INTERFACE ITF_SaMController EXTENDS ITF_BaseControlElement, ITF_SaMControllerConfigure, ITF_SaMControllerCommandChange, ITF_BaseSaM

METHOD Execute : BOOL
VAR_INPUT
	iNumberOfCommand		: INT;
	eChangeCategory			: E_SaMChangeCategory;
END_VAR
END_METHOD

METHOD ExecuteTopElementOperationsForCurrentState : BOOL
VAR_INPUT
	itfTopElement				: ITF_BaseSaMStateMethod;
END_VAR
END_METHOD

METHOD PUBLIC ExitActivState
VAR_INPUT
END_VAR
END_METHOD

METHOD PUBLIC GetActiveModeName : ST_BaseLabel
VAR_INPUT
END_VAR
END_METHOD

METHOD PUBLIC GetActiveStateName : ST_BaseLabel
VAR_INPUT
END_VAR
END_METHOD

METHOD PUBLIC GetMode : E_BaseMachineMode
VAR_INPUT
END_VAR
END_METHOD

METHOD PUBLIC GetModeName : ST_BaseLabel
VAR_INPUT
	iNumber			: INT;
END_VAR
END_METHOD

METHOD PUBLIC GetState : E_BaseMachineState
VAR_INPUT
END_VAR
END_METHOD

METHOD GetStateName : ST_BaseLabel
VAR_INPUT
	iNumber			: INT;
END_VAR
END_METHOD

METHOD PUBLIC GetTimeStateForCurrentMode : LTIME
VAR_INPUT
	iNumber		: INT;
END_VAR
END_METHOD

METHOD PUBLIC GetTimeStateForMode : LTIME
VAR_INPUT
	iMode		: int;
	iState		: INT;
END_VAR
END_METHOD

METHOD PUBLIC GetTimeWorkForMode : LTIME
VAR_INPUT
	iMode	: INT;
END_VAR
END_METHOD

METHOD PUBLIC IncrementTimeStateAndMode
VAR_INPUT
	tInterval				: TIME := T#100MS;
END_VAR
END_METHOD

METHOD PUBLIC IsChangeModeBusy : BOOL
VAR_INPUT
END_VAR
END_METHOD

METHOD PUBLIC IsChangeModeDone : BOOL
VAR_INPUT
END_VAR
END_METHOD

METHOD PUBLIC IsChangeModeStatus : BOOL
VAR_INPUT
END_VAR
END_METHOD

METHOD PUBLIC IsChangeStateBusy : BOOL
VAR_INPUT
END_VAR
END_METHOD

METHOD PUBLIC IsChangeStateDone : BOOL
VAR_INPUT
END_VAR
END_METHOD

METHOD PUBLIC IsChangeStateStatus : BOOL
VAR_INPUT
END_VAR
END_METHOD

(*			
	RafalOS
	Rafał Osajda		25.11.2025		TC 4024.66
	Zwraca czy tryb o podanym numerze jest włączony
*)
METHOD IsModeEnabled : BOOL
VAR_INPUT
	iMode 	: INT;
END_VAR
END_METHOD

(*			
	RafalOS
	Rafał Osajda		25.11.2025		TC 4024.66
	Informacja czy zadany stan jest stanem aktualnym
*)
METHOD PUBLIC IsStateIsActual : BOOL
VAR_INPUT
	iTestState	: INT;
END_VAR
END_METHOD

METHOD PUBLIC IsStateTypeActive : BOOL
VAR_INPUT
END_VAR
END_METHOD

END_INTERFACE

(* stored: Version 1.1.0.1
   Itf ITF_SaMController: Id {c7f4a38b-e5fc-0e2c-38d0-203cc4e95405}
   Method Execute: Id {63ca3afc-c287-0bdd-12ae-e0974b7b3d54}
   Method ExecuteTopElementOperationsForCurrentState: Id {39fee9f5-3dd7-0b11-0632-2982610ba37f}
   Method ExitActivState: Id {cb9e97a3-d22a-0cd9-02f4-6cb8ea8c3bb2}
   Method GetActiveModeName: Id {3dc9f8c2-6c57-0264-38ab-ef4a4f7dd9aa}
   Method GetActiveStateName: Id {838c51ac-28c2-0b15-14b8-5b0e11943641}
   Method GetMode: Id {1d69f223-181f-0972-3ad1-54d77ed4be14}
   Method GetModeName: Id {91319612-614a-053b-3f6c-986b697b0680}
   Method GetState: Id {b839727c-3386-0559-0733-9b44c3817a01}
   Method GetStateName: Id {80d7bc49-b3dd-01a8-2327-4eb12ee1406b}
   Method GetTimeStateForCurrentMode: Id {9ff2f103-5ceb-04bb-3b3e-33be3a04971a}
   Method GetTimeStateForMode: Id {240537f6-f716-06dd-2c19-f55d1c681a4f}
   Method GetTimeWorkForMode: Id {04f77d6d-980c-0fce-394f-46439c904b37}
   Method IncrementTimeStateAndMode: Id {fdc75c55-8250-02e9-11c9-c3b0fb9c4e0b}
   Method IsChangeModeBusy: Id {73bde51a-f1cb-03c3-05cb-d231e41b8173}
   Method IsChangeModeDone: Id {aa2a3fdb-2759-03f4-0561-42f93974f928}
   Method IsChangeModeStatus: Id {e91da177-da6e-070f-13f5-9d907fb4dad3}
   Method IsChangeStateBusy: Id {2c3ca8da-7edb-06c9-2406-8ed89d3c1841}
   Method IsChangeStateDone: Id {613c6918-490c-0d09-051a-6b090bdae6b4}
   Method IsChangeStateStatus: Id {65896b9c-a764-034c-3270-ababbefc1d46}
   Method IsModeEnabled: Id {97697320-58ea-077e-2495-b550560ba254}
   Method IsStateIsActual: Id {e89a67a0-e9a4-0e36-2b43-8fa5f6d48d06}
   Method IsStateTypeActive: Id {e84694eb-2fa3-0f44-1c4e-04cf04acd99f} *)
